// TwinCAT 3 PLC project mobject_errors
// Title: mobject-errors
// Company: mobject
// Author: mobject dev team
// ProjectVersion: 0.3.0
// ProgramVersion: 3.1.4024.0
// libraries:
//   Tc2_System, * (Beckhoff Automation GmbH)
//   mobject-disposable,1.1.1,mobject
//   mobject-serialization,0.5.0,mobject
// project tree:
//   Errors/ Error.TcPOU, NullError.TcPOU
//   Interfaces/ I_Error.TcIO, I_ErrorVisitor.TcIO

// ---- Interfaces/I_Error.TcIO
INTERFACE I_Error EXTENDS I_Serializable, I_Disposable

METHOD PUBLIC Accept
VAR_INPUT
	Visitor : I_ErrorVisitor;
END_VAR
END_METHOD

PROPERTY ErrorType : T_MAXSTRING
GET
END_GET
END_PROPERTY

METHOD PUBLIC IsSameAs : BOOL
VAR_INPUT
	Error : I_Error;
END_VAR
END_METHOD

PROPERTY Message : T_MAXSTRING
GET
END_GET
END_PROPERTY

END_INTERFACE

// ---- Interfaces/I_ErrorVisitor.TcIO
INTERFACE I_ErrorVisitor

METHOD VisitError
VAR_INPUT
	VisitingError : I_Error;
END_VAR
END_METHOD

END_INTERFACE

// ---- Errors/Error.TcPOU
{attribute 'linkalways'} 
{attribute 'no_explicit_call' := 'This FB is a CLASS and must be accessed using methods or properties'}
{attribute 'enable_dynamic_creation'}
FUNCTION_BLOCK ABSTRACT Error EXTENDS Disposable IMPLEMENTS I_Error
VAR
END_VAR

METHOD PUBLIC Accept
VAR_INPUT
	Visitor : I_ErrorVisitor;
END_VAR
Visitor.VisitError(THIS^);
END_METHOD

PROPERTY PUBLIC ABSTRACT ErrorType : T_MAXSTRING
GET
END_GET
END_PROPERTY

METHOD PUBLIC IsSameAs : BOOL
VAR_INPUT
	Error : I_Error;
END_VAR
IF Error = 0 THEN
	RETURN;
END_IF

IF Error.ErrorType <> THIS^.ErrorType THEN
	RETURN;
END_IF

IsSameAs := TRUE;
END_METHOD

PROPERTY PUBLIC ABSTRACT Message : T_MAXSTRING
GET
END_GET
END_PROPERTY

METHOD PROTECTED OnSerialize
VAR_INPUT
	Serializer : I_Serializer;
END_VAR
END_METHOD

METHOD PUBLIC SerializeWith
VAR_INPUT
	Serializer : I_Serializer;
END_VAR
Serializer.StartObject();
Serializer.AddKeyString('errorType',ErrorType);
Serializer.AddKeyString('message',Message);
OnSerialize(Serializer);
Serializer.EndObject();
END_METHOD

END_FUNCTION_BLOCK

// ---- Errors/NullError.TcPOU
{attribute 'linkalways'} 
{attribute 'no_explicit_call' := 'This FB is a CLASS and must be accessed using methods or properties'}
{attribute 'enable_dynamic_creation'}
FUNCTION_BLOCK NullError EXTENDS Error
VAR
END_VAR

PROPERTY ErrorType : T_MAXSTRING
GET
END_GET
END_PROPERTY

PROPERTY PUBLIC Message : T_MAXSTRING
GET
END_GET
END_PROPERTY

METHOD PUBLIC SerializeWith
VAR_INPUT
	Serializer : I_Serializer;
END_VAR
END_METHOD

END_FUNCTION_BLOCK
